FUNCTION_BLOCK Ventosa (* Template for a Basic Function Block Type *)
  (* Standard: 61499-2 *)
  (* Version 1.0, 2025-02-05, Bruno *)
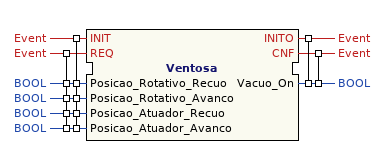
  EVENT_INPUT
    INIT WITH Posicao_Rotativo_Recuo, Posicao_Rotativo_Avanco, Posicao_Atuador_Recuo, Posicao_Atuador_Avanco; (* Initialization Request *)
    REQ WITH Posicao_Rotativo_Recuo, Posicao_Rotativo_Avanco, Posicao_Atuador_Recuo, Posicao_Atuador_Avanco; (* Normal Execution Request *)
  END_EVENT
  EVENT_OUTPUT
    INITO WITH Vacuo_On; (* Initialization Confirm *)
    CNF WITH Vacuo_On; (* Execution Confirmation *)
  END_EVENT
  VAR_INPUT
    Posicao_Rotativo_Recuo : BOOL; (* Input event qualifier *)
    Posicao_Rotativo_Avanco : BOOL;
    Posicao_Atuador_Recuo : BOOL;
    Posicao_Atuador_Avanco : BOOL;
  END_VAR
  VAR_OUTPUT
    Vacuo_On : BOOL; (* Output event qualifier *)
  END_VAR
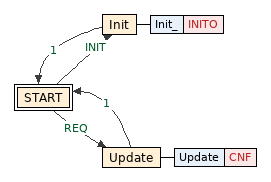
  EC_STATES
    START; (* Initial State *)
    Init : Init_ -> INITO;
    Update : Update -> CNF;
  END_STATES
  EC_TRANSITIONS
    START TO Init := INIT;
    START TO Update := REQ;
    Update TO START := 1;
    Init TO START := 1;
  END_TRANSITIONS
  ALGORITHM Init_ IN ST:
Vacuo_On:=TRUE;
  END_ALGORITHM
  ALGORITHM Update IN ST:
Vacuo_On:=TRUE;

IF Posicao_Rotativo_Recuo THEN

Vacuo_On:=FALSE;

END_IF;
  END_ALGORITHM
END_FUNCTION_BLOCK
